{attribute 'GeneratedUsingTerminal: Flexi Soft EtherCAT Gateway-0000-0001'}
{attribute addProperty BoxType "Flexi Soft EtherCAT Gateway-0000-0001"}
{attribute addProperty Id "DiagAT %I*USINT1In_Dataset1AT %I*ARRAY [0..9] OF BYTE0In_Dataset2AT %I*ARRAY [0..9] OF BYTE0In_Dataset3AT %I*ARRAY [0..9] OF BYTE0In_Dataset4AT %I*ARRAY [0..9] OF BYTE0In_Dataset5AT %I*ARRAY [0..9] OF BYTE0"}
{attribute addProperty CRC "949956373"}
{attribute addProperty Size "1"}
TYPE In_389F2F15 EXTENDS TcoIo.InputBase_8311D824 :
STRUCT
	{attribute addProperty Name "Diag"}
	Diag AT %I* : USINT;
	{attribute addProperty Name "In_Dataset1"}
	In_Dataset1 AT %I* : ARRAY [0..9] OF BYTE;
	{attribute addProperty Name "In_Dataset2"}
	In_Dataset2 AT %I* : ARRAY [0..9] OF BYTE;
	{attribute addProperty Name "In_Dataset3"}
	In_Dataset3 AT %I* : ARRAY [0..9] OF BYTE;
	{attribute addProperty Name "In_Dataset4"}
	In_Dataset4 AT %I* : ARRAY [0..9] OF BYTE;
	{attribute addProperty Name "In_Dataset5"}
	In_Dataset5 AT %I* : ARRAY [0..9] OF BYTE;
END_STRUCT
END_TYPE

(* stored: Version 1.2.0.0, ProductVersion 3.1.4024.11
   DUT In_389F2F15: Id {2b70ad14-75a7-00c5-2173-b5c427862b08} *)
